FUNCTION_BLOCK fb_safety
VAR_INPUT
	bPower    : BOOL; // Turn on motor
	bReset    : BOOL; // Error reset
	bHalt     : BOOL; // Halt button pressed
	bSeqHalt  : BOOL; // Halt from movement controler
	bHome     : BOOL; // Start homing seq
	bEndStopH : BOOL; // Physical endstop max
	bEndStopL : BOOL; // Physical endstop 0
END_VAR

VAR_OUTPUT
	bPowerStatus : BOOL; // Power on 
	bHaltDone    : BOOL; // Motor stopped
END_VAR

VAR
	// Safety FBs
    fbMC_Power  : MC_Power;
    fbMC_Reset	: MC_Reset;
	fbMC_Halt	: MC_Halt;
	
	// Homing
	fbMC_Homing : MC_Home;

	// Edge detection
	rtResetTrigger : R_TRIG;
	rtHome         : R_TRIG;
	
	// Halt help variable
	bMainHalt     : BOOL;
	
	// Power help variables
	bPowerBusy    : BOOL;
	bPowerError   : BOOL;
	nPowerErrorID : UDINT;
	bPowerPos     : BOOL;
	bPowerNeg     : BOOL;
END_VAR

VAR_IN_OUT
	stAxis   : Axis_REF; 
END_VAR


///////////////////////
// Main safety logic //
///////////////////////

// Start homing sequence
rtHome(CLK := bHome);

fbMC_Homing(
	Axis:= stAxis, 
	Execute:= rtHome.Q, 
	Position:= 0.0, 
	HomingMode:= MC_DefaultHoming, 
	bCalibrationCam:= bEndStopL);
	
// endstops logic
IF fbMC_Homing.Busy THEN
    bPowerPos := bPower;
    bPowerNeg := bPower;
ELSE
    bPowerPos := bPower AND NOT bEndStopH;
    bPowerNeg := bPower AND NOT bEndStopL;
END_IF

// Power on axis
fbMC_Power(
    Axis:= stAxis,
    Enable:= bPower,
    Enable_Positive:= bPowerPos,
    Enable_Negative:= bPowerNeg,
    Override:= 100.0);

// Reset axis errors
rtResetTrigger(CLK := bReset);
fbMC_Reset( 
	Axis := stAxis,
	Execute := rtResetTrigger.Q);
	
// Stop movement
bMainHalt := bHalt OR bSeqHalt;

fbMC_Halt(
	Axis := stAxis, 
	Execute := bMainHalt);
	
/////////////////////
// Status outputts //
/////////////////////

// Power status
bPowerStatus := fbMC_Power.Status;
bPowerBusy := fbMC_Power.Busy;
bPowerError := fbMC_Power.Error;
nPowerErrorID := fbMC_Power.ErrorID;

// Homing status (TODO)

// Check if motor stoped
bHaltDone := fbMC_Halt.Done;

END_FUNCTION_BLOCK

(* stored: Version 1.1.0.1, ProductVersion 3.1.4024.15
   POU fb_safety: Id {2b1a91eb-6451-41aa-b214-38ff110b08ec}, SpecialFunc None *)
